// TIA Portal V21 export
TYPE "Rcp_Name_Type"
TITLE = Parte Generica Della Ricetta
   STRUCT
      "Name" : String[30];
   END_STRUCT;
END_TYPE
